INTERFACE I_Observer

METHOD Update : BOOL
VAR_INPUT
END_VAR
END_METHOD

END_INTERFACE

(* stored: Version 1.1.0.1, ProductVersion 3.1.4024.12
   Itf I_Observer: Id {de98d1d4-302a-4e6f-ba3c-1046bb2a57ee}
   Method Update: Id {a3f32625-1add-4abd-a689-749044a635c3} *)
